TYPE TcoAmsNetId :
STRUCT
    netId : ARRAY[0..5] OF BYTE;
END_STRUCT
END_TYPE

(* stored: Version 1.1.0.1, ProductVersion 3.1.4024.11
   DUT TcoAmsNetId: Id {193bb840-765a-0364-1ffe-3137d8ebf5ac} *)
